TYPE Mat76 : ARRAY[1..7, 1..6] OF LREAL; END_TYPE

(* stored: Version 1.1.0.1, ProductVersion 3.1.4024.12
   DUT Mat76: Id {9ce58231-1053-4402-b771-c2cfc408b255} *)
